FUNCTION_BLOCK FB_CNC
VAR_INPUT

END_VAR
VAR_OUTPUT
	bDone: Bool;
END_VAR
VAR
END_VAR

METHOD StartCycle : BOOL
VAR_INPUT
END_VAR
END_METHOD

END_FUNCTION_BLOCK

(* stored: Version 1.1.0.1, ProductVersion 3.1.4026.18
   POU FB_CNC: Id {beaddaaa-6ba4-41b1-8859-ef0168bd27cb}, SpecialFunc None
   Method StartCycle: Id {f7bdb1bf-f4f9-4b82-8fd3-97ff0cd58c2b} *)
